FUNCTION_BLOCK fb_CSVWrite
VAR_INPUT
	bExecute:BOOL;
	dbid:UINT;
	table:STRING(100);
END_VAR
VAR_OUTPUT
	bError:BOOL:=FALSE;
	bReady:BOOL:=FALSE;
END_VAR
VAR
	PLCDBWrite:fb_PLCDBWrite(snetid:='', tTimeout:=T#15S);
	Columnnames: ARRAY [0..4] OF STRING(50):=['Dátum', 'temp_set', 'temp_act', 'hum_set', 'hum_act'];
	InsertData:ST_InsertData;
	
	
	
END_VAR

IF bExecute THEN
	IF PLCDBWrite.WriteStruct(hDBID:=dbid,
							stablename:=table,
							pRecord:=ADR(InsertData),
							cbRecord:=SIZEOF(InsertData),
							pColumnNames:=ADR(columnNames),
							cbColumnNames:=SIZEOF(columnNames))
	THEN
	IF plcdbwrite.bError THEN
		bError:=TRUE;
		
	ELSE 
	IF NOT plcdbwrite.bBusy THEN
		bExecute:=FALSE;
		bReady:=TRUE;
	END_IF
	END_IF
END_IF	
	
							
END_IF

METHOD Reset : BOOL
VAR_INPUT
END_VAR
BReady:=false;
END_METHOD

END_FUNCTION_BLOCK

(* stored: Version 1.1.0.1, ProductVersion 3.1.4024.2
   POU fb_CSVWrite: Id {f0c3ef67-6118-4832-9964-b88959bf2466}, SpecialFunc None
   Method Reset: Id {816436ef-fd9c-44c2-8646-92722839c530} *)
